TEXTLIST CoEParamTextList
  1 = 'Maximal Current'
  2 = 'Reduced Current'
  3 = 'Nominal Voltage'
  4 = 'Motor Coil Resistance'
  6 = 'Full steps'
  10 = 'Motor Coil Inductance'
   = ''
END_TEXTLIST

(* stored: Version 1.1.0.1
   TextList CoEParamTextList: Id {4d9ffcd1-7a68-40dc-b979-fbaf840b8192} *)
